FUNCTION_BLOCK fbLdConveyor3Zones
VAR_INPUT

	bEnable		: BOOL;
	bRapidPB	: BOOL;
	bLdBasketZone1TransferMemoryBit: BOOL;
	bLdBasketZone1ConfirmMemoryBit: BOOL;
	bLdBasketZone2TransferMemoryBit: BOOL;
	bLdBasketZone2ConfirmMemoryBit	: BOOL;

	bLdSensor1: BOOL;
	bLdSensor2: BOOL;
	bLdEndSensor: BOOL;

	diZone1BasketConfirmDelayTime	: DINT;

(*	diZone2BasketConfirmDelayTime	: DINT;
	diRapidPBDelayTime	: DINT;
*)
	diEndZoneBasketConfirmDelayTime	: DINT;

	bEmergencyStop: BOOL;
END_VAR
VAR_OUTPUT
	bMotorOnOff	: BOOL;
END_VAR
VAR
	bRapidPBRE: R_TRIG;
	bMotorStopBit: BOOL;
	TON1: TON;
	TON2: TON;
	bConvAutoCut: BOOL;
	tLdZone1SensorDelayTime: TON;

	(*TRIG1: R_TRIG;
	Trig2: R_TRIG;
	TON3: TON;
	RampIn: BOOL;
	TON4: TON;
	CVDelayOff : BOOL;
	TON5: TON;*)

END_VAR

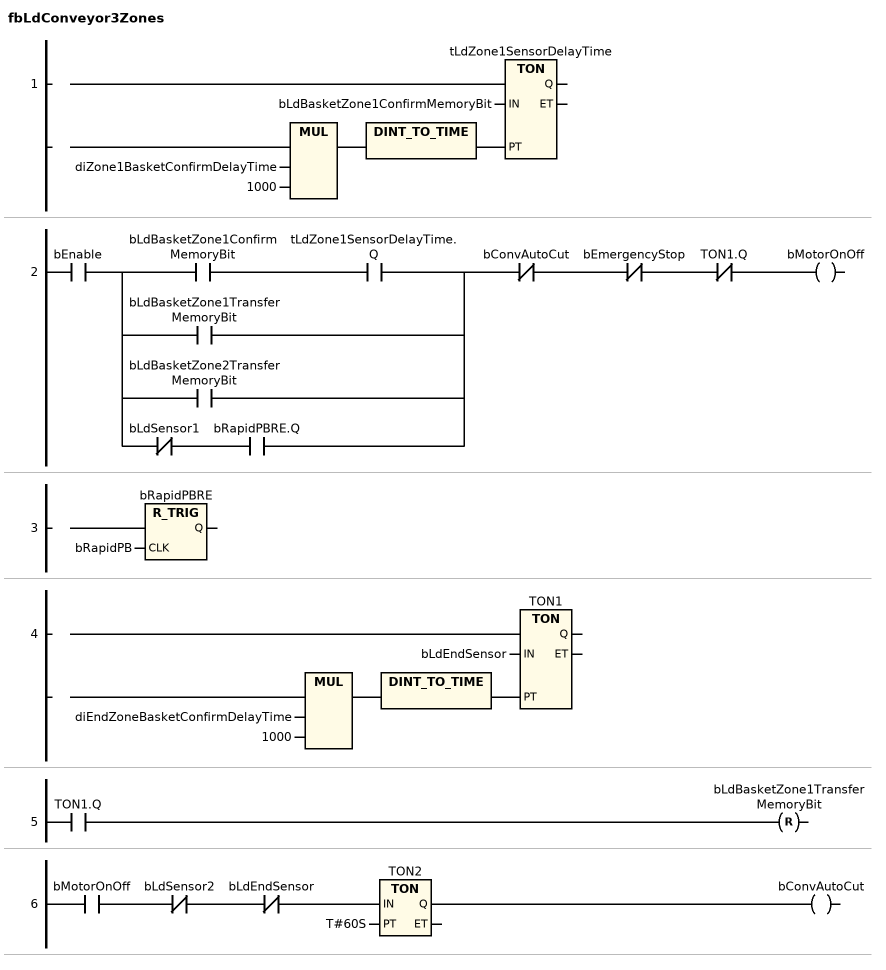
// NETWORK 1
tLdZone1SensorDelayTime(IN := bLdBasketZone1ConfirmMemoryBit, PT := DINT_TO_TIME(diZone1BasketConfirmDelayTime * 1000)); // TON

// NETWORK 2
bMotorOnOff := (bEnable AND (bLdBasketZone1ConfirmMemoryBit AND tLdZone1SensorDelayTime.Q OR bLdBasketZone1TransferMemoryBit OR bLdBasketZone2TransferMemoryBit OR NOT bLdSensor1 AND bRapidPBRE.Q)) AND NOT bConvAutoCut AND NOT bEmergencyStop AND NOT TON1.Q;

// NETWORK 3
bRapidPBRE(CLK := bRapidPB); // R_TRIG

// NETWORK 4
TON1(IN := bLdEndSensor, PT := DINT_TO_TIME(diEndZoneBasketConfirmDelayTime * 1000)); // TON

// NETWORK 5
bLdBasketZone1TransferMemoryBit R= TON1.Q;

// NETWORK 6
TON2(IN := bMotorOnOff AND NOT bLdSensor2 AND NOT bLdEndSensor, PT := T#60S); // TON
bConvAutoCut := TON2.Q;

END_FUNCTION_BLOCK

(* stored: Version 1.1.0.1, ProductVersion 3.1.4024.12
   POU fbLdConveyor3Zones: Id {deef62da-9c2e-4ab5-adca-c6dc5250ea0f}, SpecialFunc None *)
